{attribute 'linkalways'} 
{attribute 'no_explicit_call' := 'This FB is a CLASS and must be accessed using methods or properties'}
{attribute 'enable_dynamic_creation'}
FUNCTION_BLOCK Node_F_VN_UprightBoundingRectangle EXTENDS VisionNode
VAR
    ipPointSet : _ITcVnContainer;
    stRectangle : _TcVnRectangle_UDINT;
    hrPrev : _HRESULT(S_OK);
	hresult : _HRESULT(S_OK);
END_VAR

METHOD PUBLIC  Clone : I_Node
VAR
	pNode : POINTER TO Node_F_VN_UprightBoundingRectangle;
END_VAR
pNode := __NEW(Node_F_VN_UprightBoundingRectangle);
Clone := pNode^;
END_METHOD

METHOD FB_init : BOOL
VAR_INPUT
	bInitRetains : BOOL; // if TRUE, the retain variables are initialized (warm start / cold start)
	bInCopyCode : BOOL;  // if TRUE, the instance afterwards gets moved into the copy code (online change)
END_VAR
AddInput('ipPointSet', ipPointSet);
AddInput('hrPrev', hrPrev);
AddOutput('stRectangle', stRectangle);
AddOutput('hresult',hresult);
END_METHOD

METHOD PROTECTED OnExecute
hresult.Value := F_VN_UprightBoundingRectangle(
	ipPointSet := ipPointSet.Value,
    stRectangle := stRectangle.Value,
	hrPrev:= hrPrev.Value);
END_METHOD

METHOD PUBLIC PreExecutionCheck
VAR_INPUT
	Check : I_PreExecutionChecks;
END_VAR
Check.IsTrue(ipPointSet.IsValid, 'ipPointSet must be a valid container');
Check.IsTrue((ipPointSet.IsType(TC_GLOBAL_CONST_LIST.ContainerType_Vector_TcVnPoint2_DINT) OR
              ipPointSet.IsType(TC_GLOBAL_CONST_LIST.ContainerType_Vector_TcVnPoint2_REAL)),
              'ipPointSet contains incorrect type');
END_METHOD

END_FUNCTION_BLOCK

(* stored: Version 1.1.0.1, ProductVersion 3.1.4026.13
   POU Node_F_VN_UprightBoundingRectangle: Id {6872f937-4404-0e00-16be-c645c7550c75}, SpecialFunc None
   Folder Constructor: Id {63c182f8-92c9-05db-1dc4-6f80f73cacd2}
   Method Clone: Id {acb8f266-6f8f-0864-12bf-ccff3555e437}
   Method FB_init: Id {eda51280-9b55-0883-23df-70119f90c56b}
   Method OnExecute: Id {e5955091-a07d-0e52-1278-aa663c99dc16}
   Method PreExecutionCheck: Id {e4926c8a-9938-065d-108a-f0cdcb9fb725} *)
